TYPE U_AXIS_CTRL :
UNION

  stCtrl              : ARRAY[1..MAX_AXIS] OF ST_AXIS_CTRL;

  byCtrl    AT %I*    : ARRAY[1..MAX_AXIS] OF
                        ARRAY[1..SIZEOF(ST_AXIS_CTRL)] OF BYTE;
END_UNION
END_TYPE

(* stored: Version 1.1.0.1, ProductVersion 3.1.4026.13
   DUT U_AXIS_CTRL: Id {6f5d7241-97df-0c04-2491-c9b14687d6f4} *)
